# EPICS substitutions: lensApp/Db/flexiblelimit.substitutions
file flexiblelimit.tpl-db
{
    {
        LOCATION = $(LOCATION)
        LIMIT    = $(LIMIT)
        SIDE     = $(SIDE)
        TYPE     = $(TYPE)
    }
}
